// TIA Portal V20 export
DATA_BLOCK "Simulation_DB"   // DB3
// stored: InstanceOfName Unit1.Em0.Simulation, InstanceOfType FB, Namespace Unit1.Em0
"Unit1.Em0.Simulation"
   // VAR_INPUT
   //    simulation : Bool;
   // END_VAR
   // VAR
   //    instActuator { ExternalAccessible := 'False'; ExternalVisible := 'False'; ExternalWritable := 'False'} : Array[0..9] of "Simulation_Actuator";
   // END_VAR
BEGIN
END_DATA_BLOCK
